{attribute 'linkalways'} 
{attribute 'no_explicit_call' := 'This FB is a CLASS and must be accessed using methods or properties'}
{attribute 'enable_dynamic_creation'}
FUNCTION_BLOCK _TcVnVector4_LREAL EXTENDS AliasDatatypeBase
VAR
	localData : TcVnVector4_LREAL;
	activeData : REFERENCE TO TcVnVector4_LREAL REF= localData;
	aliasBaseDatatype : _Array0to3OfLREAL;
END_VAR

PROPERTY PUBLIC Address : PVOID
GET
Address := ADR(activeData);
END_GET
END_PROPERTY

METHOD PUBLIC ClearReference
VAR_INPUT
END_VAR
activeData REF= localData;
SetBaseDatatypeReference();
END_METHOD

METHOD PUBLIC Clone : I_Datatype
VAR
    pClone : POINTER TO _TcVnVector4_LREAL;
END_VAR
pClone := __NEW(_TcVnVector4_LREAL);
Clone := pClone^;
END_METHOD

METHOD FB_init : BOOL
VAR_INPUT
	bInitRetains : BOOL; // if TRUE, the retain variables are initialized (warm start / cold start)
	bInCopyCode : BOOL;  // if TRUE, the instance afterwards gets moved into the copy code (online change)
	//InitialValue : <type>; // if possible, not all values can be initialized
END_VAR
//localData := InitialValue; // if possible, not all values can be initialized
SetBaseDatatypeReference();
AddBaseDatatype(aliasBaseDatatype);
END_METHOD

PROPERTY PUBLIC Identifier : T_MAXSTRING
GET
Identifier := 'TcVnVector4_LREAL';
END_GET
END_PROPERTY

METHOD PUBLIC MakeReferenceTo
VAR_INPUT
	ReferenceTarget : REFERENCE TO TcVnVector4_LREAL;
END_VAR
activeData REF= ReferenceTarget;
SetBaseDatatypeReference();
END_METHOD

METHOD PROTECTED SetBaseDatatypeReference
VAR_INPUT
END_VAR
aliasBaseDatatype.MakeReferenceTo(activeData);
END_METHOD

PROPERTY PUBLIC Size : UDINT
GET
Size := SIZEOF(activeData);
END_GET
END_PROPERTY

METHOD TryMakeReferenceTo : BOOL
VAR_INPUT
	Target : I_Datatype;
END_VAR
VAR
	pTargetData : POINTER TO TcVnVector4_LREAL;
END_VAR
IF NOT IsEquivalentTo(Target) THEN
	RETURN;
END_IF

pTargetData := Target.Address;
activeData REF= pTargetData^;
SetBaseDatatypeReference();
TryMakeReferenceTo := TRUE;
END_METHOD

PROPERTY PUBLIC Value : REFERENCE TO TcVnVector4_LREAL
GET
Value REF= activeData;
END_GET
END_PROPERTY

END_FUNCTION_BLOCK

(* stored: Version 1.1.0.1, ProductVersion 3.1.4024.13
   POU _TcVnVector4_LREAL: Id {7edd440f-66f2-06ac-2565-b22a90f99933}, SpecialFunc None
   Folder Core: Id {d2e20909-6374-07f7-3377-b74ce36cc857}
   Folder Protected: Id {4bbdea95-f945-0707-10e8-18ab6a7720d8}
   Folder Customize: Id {96b5f36a-d9bd-0d07-2212-e08b56ed22f7}
   Folder Constructor: Id {f97c1c17-cd83-0f1d-04b6-5de64e4ec8c6}
   Property Address: Id {2bace0f8-2305-0564-1ca3-014f8043d9f9}
   Get Get: Id {2b68826d-f87c-0da4-3690-7caae3b3ce49}
   Method ClearReference: Id {37fa3e28-a04e-059e-1377-6f7092419472}
   Method Clone: Id {88df8090-cc41-02d6-143f-b358af17b5d7}
   Method FB_init: Id {48a28009-9ab1-0f1e-2e72-7deb6f2ccca3}
   Property Identifier: Id {17e75cbf-8578-0641-0f18-9f721922a19f}
   Get Get: Id {0752cda2-bcc1-0eca-3817-5576d014ec3c}
   Method MakeReferenceTo: Id {b2788ebe-b9a0-0059-1482-8bb21a5e127f}
   Method SetBaseDatatypeReference: Id {90f67ce4-a16a-0dc1-2cc9-51dbfc0d4a4a}
   Property Size: Id {ecc4608c-3f96-097a-2cdc-6455ec603edb}
   Get Get: Id {23d8ba8f-21da-03ef-19b4-0f3df70487fa}
   Method TryMakeReferenceTo: Id {3b554658-8acf-0756-2fe0-f2e907fedde2}
   Property Value: Id {f9203bdd-e2d2-0ee0-3b00-046a6532fefc}
   Get Get: Id {b88d1e04-11f0-024c-1220-748d2140957f} *)
